FUNCTION_BLOCK earth_fault_1 (* Composite Function Block Type *)
  (* Standard: 61499-2 *)
  (* Version 0.0, 3/23/2016, gulzha, nxtControl GmbH, template *)
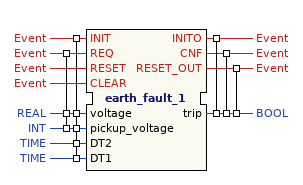
  EVENT_INPUT
    INIT WITH pickup_voltage, voltage, DT1, DT2; (* Initialization Request *)
    REQ WITH pickup_voltage, voltage; (* Normal Execution Request *)
    RESET;
    CLEAR;
  END_EVENT
  EVENT_OUTPUT
    INITO WITH trip; (* Initialization Confirm *)
    CNF WITH trip; (* Execution Confirmation *)
    RESET_OUT WITH trip;
  END_EVENT
  VAR_INPUT
    voltage : REAL;
    pickup_voltage : INT;
    DT2 : TIME; (* Delay Time *)
    DT1 : TIME; (* Delay Time *)
  END_VAR
  VAR_OUTPUT
    trip : BOOL;
  END_VAR
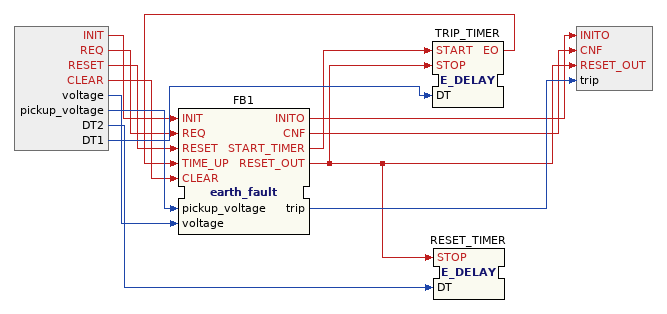
  FBS
    TRIP_TIMER : E_DELAY;
    RESET_TIMER : E_DELAY;
    FB1 : earth_fault;
  END_FBS
  EVENT_CONNECTIONS
    INIT TO FB1.INIT;
    REQ TO FB1.REQ;
    RESET TO FB1.RESET;
    TRIP_TIMER.EO TO FB1.TIME_UP;
    CLEAR TO FB1.CLEAR;
    FB1.INITO TO INITO;
    FB1.CNF TO CNF;
    FB1.START_TIMER TO TRIP_TIMER.START;
    FB1.RESET_OUT TO TRIP_TIMER.STOP;
    FB1.RESET_OUT TO RESET_TIMER.STOP;
    FB1.RESET_OUT TO RESET_OUT;
  END_CONNECTIONS
  DATA_CONNECTIONS
    DT1 TO TRIP_TIMER.DT;
    DT2 TO RESET_TIMER.DT;
    pickup_voltage TO FB1.pickup_voltage;
    voltage TO FB1.voltage;
    FB1.trip TO trip;
  END_CONNECTIONS
END_FUNCTION_BLOCK
